PROGRAM MAIN
VAR
	bButton : BOOL;
END_VAR

P_TrackRemainingTime();
P_LoginFromPLC();
P_ListUsers();

END_PROGRAM

(* stored: Version 1.1.0.1, ProductVersion 3.1.4024.3
   POU MAIN: Id {be712938-f49c-4500-970d-9ea04678be54}, SpecialFunc None *)
